//{attribute 'pack_mode' := '8'}
TYPE ST_PCMSettings :
STRUCT
	ToleranceThresholdPK		:	ST_ToleranceThresholdPK;
	ToleranceThresholdOUT		:	ST_ToleranceThresholdOUT;
	ToleranceThresholdCS		:	ST_ToleranceThresholdCS;
END_STRUCT
END_TYPE

(* stored: Version 1.1.0.1
   DUT ST_PCMSettings: Id {a65ddeeb-96f9-412b-9c0c-540a5cbf55da} *)
